FUNCTION_BLOCK FN_2_2_Finite_State_Machine

VAR CONSTANT
	MIXERDURATION : TIME := T#5S;
	PUMPDURATION  : TIME := T#3S;
	GATEDURATION  : TIME := T#2S;	
END_VAR

VAR_INPUT
	startPB : BOOL;
	stopPB : BOOL;
END_VAR

VAR_OUTPUT
	mixerState : BOOL;
	pumpState  : BOOL;
	gateState  : BOOL;
END_VAR

VAR
	startTrig : R_TRIG;
	stopTrig  : R_TRIG;

	state : (init, mixerON, pumpON, gateOpen, close);

	timer : TON;
END_VAR

stopTrig(CLK := stopPB);

IF NOT stopPB THEN // Ensure Stop PB is not pressed before checking startPB
	startTrig(CLK := startPB);
END_IF

CASE state OF
	init : // default state
		IF startTrig.Q THEN
			state := mixerON;
		END_IF
	
	mixerON: // Turn ON mixer for MIXERDURATION[default 5s]
		mixerState := TRUE;
		timer(IN := TRUE, PT := MIXERDURATION);	
		IF timer.Q THEN
			timer(IN := FALSE);
			state := pumpON;
		END_IF
	
	pumpON: // Turn ON pump for PUMPDURATION[default 4s]
		pumpState := TRUE;
		timer(IN := TRUE, PT := PUMPDURATION);	
		IF timer.Q THEN
			pumpState := FALSE;
			timer(IN := FALSE);
			state := gateOpen;
		END_IF
	
	gateOpen: // Open gate for GATEDURATION[default 3s]
		timer(IN := TRUE, PT := GATEDURATION);	
		IF timer.Q THEN
			timer(IN := FALSE);
			state := close;
		END_IF
	
	close: // Tidy up variables and loop to start
		M_resetvariables();
		state := init;
END_CASE

IF stopTrig.Q THEN
	state := close;
END_IF

METHOD PRIVATE M_resetvariables : BOOL
VAR_INPUT
END_VAR
timer(IN := FALSE);	
mixerState := FALSE;
pumpState := FALSE;
gateState := FALSE;
END_METHOD

END_FUNCTION_BLOCK

(* stored: Version 1.1.0.1, ProductVersion 3.1.4024.13
   POU FN_2_2_Finite_State_Machine: Id {4c9a9bc5-5333-4a3f-bcb2-f1df696691b8}, SpecialFunc None
   Method M_resetvariables: Id {a186e712-bf97-49c5-abe2-9780c4790c37} *)
